(* IEC 61131-3 sources: RL_MAR/experiments/comparison/autoplc/results/gpt-4o_20260511_211137/med_70, 1 file *)

(* ---- med_70_1.st ---- *)
FUNCTION_BLOCK EggIncubatorControl
    VAR_INPUT
        StartButton : BOOL; (* Input for starting the incubation process *)
        StopButton : BOOL; (* Input for stopping the incubation process *)
        TemperatureSensor : REAL; (* Input for temperature reading in °C *)
        HumiditySensor : REAL; (* Input for humidity reading in % *)
    END_VAR

    VAR_OUTPUT
        HeatingElement : BOOL; (* Output for controlling the heating element *)
        Humidifier : BOOL; (* Output for controlling the humidifier *)
        EggTurningMotor : BOOL; (* Output for controlling the egg turning motor *)
        IncubationInProgress : BOOL; (* Indicator for an ongoing incubation process *)
    END_VAR

    VAR
        TargetTemperature : REAL; (* Target temperature in °C *)
        TargetHumidity : REAL; (* Target humidity in % *)
        TurnIntervalSeconds : INT; (* Interval for turning eggs (1 hour in seconds) *)
        TurnTimerSeconds : INT; (* Timer for egg turning cycle in seconds *)
    END_VAR

    (* Initialize control parameters *)
    TargetTemperature := 37.5;
    TargetHumidity := 50.0;
    TurnIntervalSeconds := 3600;
    TurnTimerSeconds := 0;

    (* Start/Stop Control *)
    IF StartButton AND NOT IncubationInProgress THEN
        IncubationInProgress := TRUE;
    ELSIF StopButton THEN
        IncubationInProgress := FALSE;
        HeatingElement := FALSE;
        Humidifier := FALSE;
        EggTurningMotor := FALSE;
        TurnTimerSeconds := 0;
    END_IF

    (* Temperature Control *)
    IF IncubationInProgress THEN
        IF TemperatureSensor < TargetTemperature THEN
            HeatingElement := TRUE;
        ELSE
            HeatingElement := FALSE;
        END_IF

        (* Humidity Control *)
        IF HumiditySensor < TargetHumidity THEN
            Humidifier := TRUE;
        ELSE
            Humidifier := FALSE;
        END_IF

        (* Egg Turning Cycle *)
        TurnTimerSeconds := TurnTimerSeconds + 1;
        IF TurnTimerSeconds >= TurnIntervalSeconds THEN
            EggTurningMotor := NOT EggTurningMotor;
            TurnTimerSeconds := 0;
        END_IF
    END_IF
END_FUNCTION_BLOCK
